# EPICS alarm handler configuration: mps_database/bareTest/alarms/areas/mpln_sph_mp02.alhConfig
GROUP NULL MPLN:SPH:MP02:1
$ALIAS MPS Link Node 121
$GUIDANCE
LTUH MPS
   Group Name: MPLN:SPH:MP02:1
   Summary PV:  MPLN:SPH:MP02:1:STATSUMY
$END
CHANNEL  MPLN:SPH:MP02:1    MPLN:SPH:MP02:1:MPS_EN_RBV		-----
CHANNEL  MPLN:SPH:MP02:1    MPLN:SPH:MP02:1:LC1_MODE_RBV		-----
